SUBAPPLICATION Softkey_Web_IXA (* SoftKey (VT) ODER lokaler Web-Override (vt-ui-mirror, Dauerzustand) zu 1 gemeinsamem kontinuierlichem AX-Zustand zusammengefuehrt - fuer Taster ohne AUX-Zuordnung (z.B. Fahrwerk-Mittelpunkt), die trotzdem per Web-Client genauso wie physisch gedrueckt/gehalten werden koennen sollen. Analog zu Softkey_Aux_IXA_TO_Remote_WRITE (dort zusaetzlich mit AUX + Remote-Write), hier nur der reine Merge ohne AUX und ohne Schreiben irgendwohin - der Aufrufer verarbeitet den gemergten Zustand selbst weiter (z.B. SoftKey_Kurz_Lang). *)
  (* Standard: 61499-2; Description: Copyright (c) 2026 Meisterschulen am Ostbahnhof This program and the accompanying materials are made available under the terms of the Eclipse Public License 2.0 which is available at https://www.eclipse.org/legal/epl-2.0/ SPDX-License-Identifier: EPL-2.0 *)
  (* Version 1.0, 2026-09-11, Franz Höpfinger, Meisterschulen am Ostbahnhof, initial implementation - herausgeloest aus Fahrwerk_Mittelpunkt_Automatik.SUB (Softkey_Mittelpunkt+WebSub_Mittelpunkt+OR_MITTELPUNKT), wiederverwendbar fuer jeden Taster ohne AUX, der auch per Web gehalten werden koennen soll. *)
  PACKAGE MyLib::sys;
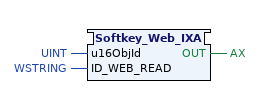
  VAR_INPUT
    u16ObjId : UINT; (* Object ID SoftKey *)
    ID_WEB_READ : WSTRING; (* Lokale Subscribe-Adresse fuer den Web-Client (vt-ui-mirror): down/up wie ein gehaltener physischer Taster *)
  END_VAR
  PLUGS
    OUT : adapter::types::unidirectional::AX; (* SoftKey ODER Web-Override, 1 gemeinsamer kontinuierlicher Zustand *)
  END_PLUGS
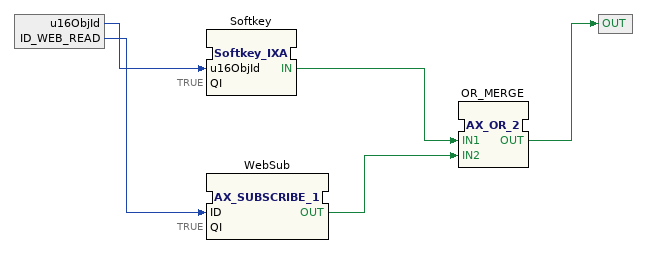
  FBS
    Softkey : isobus::UT::io::Softkey::Softkey_IXA(QI := TRUE);
    WebSub : adapter::net::AX_SUBSCRIBE_1(QI := TRUE);
    OR_MERGE : adapter::booleanOperators::AX_OR_2;
  END_FBS
  DATA_CONNECTIONS
    u16ObjId TO Softkey.u16ObjId;
    ID_WEB_READ TO WebSub.ID;
  END_CONNECTIONS
  ADAPTER_CONNECTIONS
    Softkey.IN TO OR_MERGE.IN1;
    WebSub.OUT TO OR_MERGE.IN2;
    OR_MERGE.OUT TO OUT;
  END_CONNECTIONS
END_SUBAPPLICATION
